PROGRAM MAIN
VAR
END_VAR

END_PROGRAM

(* stored: Version 1.1.0.1
   POU MAIN: Id {008be9b5-3aba-4d05-8c6f-3a468a928fa4} *)
